// TIA Portal V17 export
// export: Created 2022-07-20T06:59:44.4199644Z, ExportSetting WithDefaults, DisplayName Totally Integrated Automation Portal, DisplayVersion V17, DisplayName TIA Portal Openness, DisplayVersion V17, DisplayName TIA Portal Version Control Interface, DisplayVersion V17, DisplayName SINAMICS Startdrive Advanced, DisplayVersion V17, DisplayName SINAMICS Startdrive G130, G150, S120, S150, SINAMICS MV, S210, DisplayVersion V17, DisplayName SINAMICS Startdrive G110M, G120, G120C, G120D, G120P, G115D, DisplayVersion V17, DisplayName STEP 7 Professional, DisplayVersion V17, DisplayName STEP 7 Safety, DisplayVersion V17, DisplayName WinCC Advanced, DisplayVersion V17
FUNCTION_BLOCK "FB10076_ShutterMotorManager_1"   // FB10076, LAD
TITLE = FB10076_ShutterMotorManager_1
{ S7_Optimized_Access := 'TRUE' }
AUTHOR : Anirouddh
FAMILY : 1007x_DRYER_UV
VERSION : 1.0
// Release note : 
// 1.0 - Feature developped
// stored: AutoNumber false, IsIECCheckEnabled false, IsRetainMemResEnabled false, MemoryReserve 100, SetENOAutomatically false, UDAEnableTagReadback false
   VAR_INPUT
      ShutterMotorInError : Bool;
      PWM_PulsesSetPoint : Real;
      ShutterSensorClosed : Bool;
      RequestInitializeShutter : Bool;
      RequestOpenShutter : Bool;
      RequestCloseShutter : Bool;
      TransportActivated : Bool;
      PWMCardInError : Bool;
   END_VAR
   VAR_OUTPUT
      PWM_InitializeShutter : Bool;
      PWM_OpenShutter : Bool;
      PWM_CloseShutter : Bool;
      PWM_Pulses : Real;
      ResetPulseCard : Bool;
      ShutterError : Bool;
      ShutterInitialized : Bool;
      ShutterOpened : Bool;
      ShutterClosed : Bool;
   END_VAR
   VAR
      ShutterMovementManegement : Int;
      R_TRIG_ShutterSensorClosed { S7_SetPoint := 'True'} : R_TRIG;
      R_TRIG_RequestInitializeShutter { S7_SetPoint := 'True'} : R_TRIG;
      R_TRIG_RequestOpenShutter { S7_SetPoint := 'True'} : R_TRIG;
      R_TRIG_RequestCloseShutter { S7_SetPoint := 'True'} : R_TRIG;
      F_TRIG_TransportActivated { S7_SetPoint := 'True'} : F_TRIG;
      F_TRIG_ShutterSensorClose { S7_SetPoint := 'True'} : F_TRIG;
   END_VAR
   VAR CONSTANT
      WAIT_FOR_MOVEMENT_REQUEST : Int := 0;
      INITIALIZE_SHUTTER : Int := 10;
      OPEN_SHUTTER : Int := 20;
      CLOSE_SHUTTER : Int := 30;
      MOVEMENT_DONE : Int := 40;
      "==========" : Bool;
   END_VAR
BEGIN

REGION Network 1 (SCL): First Scan
   IF "FirstScan" THEN
       #ShutterInitialized := FALSE;
       #ShutterOpened := FALSE;
       #ShutterClosed := FALSE;
       #ShutterMovementManegement := 0;
   END_IF;
END_REGION

REGION Network 2 (SCL): Edge Signals
   REGION EDGE SIGNALS
       #R_TRIG_RequestInitializeShutter(CLK := #RequestInitializeShutter);
       #R_TRIG_RequestOpenShutter(CLK := #RequestOpenShutter);
       #R_TRIG_RequestCloseShutter(CLK := #RequestCloseShutter);
       #R_TRIG_ShutterSensorClosed(CLK := #ShutterSensorClosed);
       #F_TRIG_TransportActivated(CLK := #TransportActivated);
       #F_TRIG_ShutterSensorClose(CLK := #ShutterSensorClosed);
   END_REGION
END_REGION

REGION Network 3 (SCL): Shutter Movement Management
   CASE #ShutterMovementManegement OF
       #WAIT_FOR_MOVEMENT_REQUEST:
           IF #ShutterInitialized THEN
               IF #R_TRIG_RequestOpenShutter.Q AND #ShutterSensorClosed AND #TransportActivated THEN
                   #ShutterOpened := FALSE;
                   #ShutterClosed := FALSE;
                   #ShutterMovementManegement := #OPEN_SHUTTER;
               ELSIF (#R_TRIG_RequestCloseShutter.Q OR #F_TRIG_TransportActivated.Q) AND NOT(#ShutterSensorClosed) THEN
                   #ShutterOpened := FALSE;
                   #ShutterClosed := FALSE;
                   #ShutterMovementManegement := #CLOSE_SHUTTER;
               END_IF;
           ELSE
               IF #R_TRIG_RequestInitializeShutter.Q THEN
                   #ShutterMovementManegement := #INITIALIZE_SHUTTER;
               END_IF;
           END_IF;
       #INITIALIZE_SHUTTER:
           #PWM_InitializeShutter := TRUE;
           #PWM_Pulses := #PWM_PulsesSetPoint;
           IF #R_TRIG_ShutterSensorClosed.Q THEN
               #PWM_InitializeShutter := FALSE;
               #ShutterInitialized := TRUE;
               #ShutterOpened := FALSE;
               #ShutterClosed := TRUE;
               #ShutterMovementManegement := #MOVEMENT_DONE;
           END_IF;
       #OPEN_SHUTTER:
           #PWM_OpenShutter := TRUE;
           #PWM_Pulses := #PWM_PulsesSetPoint;
           IF #F_TRIG_ShutterSensorClose.Q THEN
               #PWM_OpenShutter := FALSE;
               #ShutterOpened := TRUE;
               #ShutterClosed := FALSE;
               #ShutterMovementManegement := #MOVEMENT_DONE;
           END_IF;
       #CLOSE_SHUTTER:
           #PWM_CloseShutter := TRUE;
           #PWM_Pulses := #PWM_PulsesSetPoint;
           IF #R_TRIG_ShutterSensorClosed.Q THEN
               #PWM_CloseShutter := FALSE;
               #ShutterOpened := FALSE;
               #ShutterClosed := TRUE;
               #ShutterMovementManegement := #MOVEMENT_DONE;
           END_IF;
       #MOVEMENT_DONE:
           #ShutterMovementManegement := #WAIT_FOR_MOVEMENT_REQUEST;
   END_CASE;
END_REGION

REGION Network 4 (SCL): Error Managament
   #ShutterError := #ShutterMotorInError;

   IF #PWMCardInError THEN
       #ResetPulseCard := TRUE;
   ELSE
       #ResetPulseCard := FALSE; 
   END_IF;
END_REGION
END_FUNCTION_BLOCK
